INTERFACE ITF_BaseFlag extends ITF_BaseFlagGet, ITF_BaseFlagSet

END_INTERFACE

(* stored: Version 1.1.0.1
   Itf ITF_BaseFlag: Id {53c74f07-99f7-0225-2af2-5711ac58b2c9} *)
